// TIA Portal V17 export
// export: Created 2023-02-14T02:49:12.4327094Z, ExportSetting WithDefaults, DisplayName Totally Integrated Automation Portal, DisplayVersion V17, DisplayName TIA Portal Openness, DisplayVersion V17, DisplayName TIA Portal Teamcenter Gateway, DisplayVersion V17, DisplayName TIA Portal Version Control Interface, DisplayVersion V17, DisplayName SINAMICS Startdrive Advanced, DisplayVersion V17, DisplayName SINAMICS Startdrive G130, G150, S120, S150, SINAMICS MV, S210, DisplayVersion V17, DisplayName SINAMICS Startdrive G110M, G120, G120C, G120D, G120P, G115D, DisplayVersion V17, DisplayName STEP 7 Professional, DisplayVersion V17, DisplayName STEP 7 Safety, DisplayVersion V17, DisplayName WinCC Professional, DisplayVersion V17
FUNCTION "Comm" : Void   // FC7, LAD
{ S7_Optimized_Access := 'TRUE' }
VERSION : 0.1
// stored: AutoNumber true, IsIECCheckEnabled false, SetENOAutomatically false, UDAEnableTagReadback false
   VAR_TEMP   // added for the SCL form of the ladder/FBD networks
      _s5time1 : S5Time;
      _s5time2 : S5Time;
      _w1 : Bool;
   END_VAR
BEGIN

REGION Network 1: THE1 Heat Beat
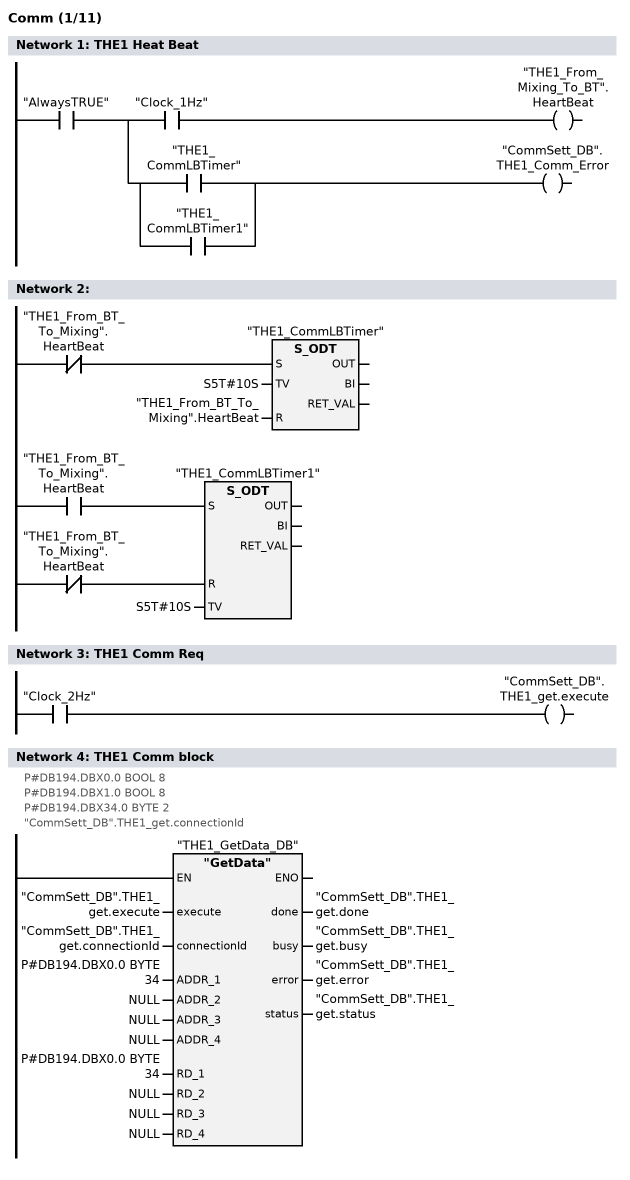
   RUNG wire#powerrail
      Contact( "AlwaysTRUE" )
      wire#w1
      Contact( "Clock_1Hz" )
      Coil( "THE1_From_Mixing_To_BT".HeartBeat )
   END_RUNG
   RUNG wire#w1
      Contact( "THE1_CommLBTimer" )
      wire#w2
      Coil( "CommSett_DB".THE1_Comm_Error )
   END_RUNG
   RUNG wire#w1
      Contact( "THE1_CommLBTimer1" )
   END_RUNG wire#w2
   // the same network as SCL:
   "THE1_From_Mixing_To_BT".HeartBeat := "AlwaysTRUE" AND "Clock_1Hz";
   "CommSett_DB".THE1_Comm_Error := "AlwaysTRUE" AND ("THE1_CommLBTimer" OR "THE1_CommLBTimer1");
END_REGION

REGION Network 2
   RUNG wire#powerrail
      I_Contact( "THE1_From_BT_To_Mixing".HeartBeat )
      S_ODT(T_NO := "THE1_CommLBTimer", TV := S5T#10S, R := "THE1_From_BT_To_Mixing".HeartBeat, BI =>, RET_VAL =>)
   END_RUNG
   RUNG wire#powerrail
      Contact( "THE1_From_BT_To_Mixing".HeartBeat )
      S_ODT(T_NO := "THE1_CommLBTimer1", R := wire#w1, TV := S5T#10S, BI =>, RET_VAL =>)
   END_RUNG
   RUNG wire#powerrail
      I_Contact( "THE1_From_BT_To_Mixing".HeartBeat )
   END_RUNG wire#w1
   // the same network as SCL:
   #_s5time1 := S_ODT(T_NO := "THE1_CommLBTimer",
                      S := NOT "THE1_From_BT_To_Mixing".HeartBeat,
                      TV := S5T#10S,
                      R := "THE1_From_BT_To_Mixing".HeartBeat);
   #_s5time2 := S_ODT(T_NO := "THE1_CommLBTimer1",
                      S := "THE1_From_BT_To_Mixing".HeartBeat,
                      R := NOT "THE1_From_BT_To_Mixing".HeartBeat,
                      TV := S5T#10S);
END_REGION

REGION Network 3: THE1 Comm Req
   RUNG wire#powerrail
      Contact( "Clock_2Hz" )
      Coil( "CommSett_DB".THE1_get.execute )
   END_RUNG
   // the same network as SCL:
   "CommSett_DB".THE1_get.execute := "Clock_2Hz";
END_REGION

REGION Network 4: THE1 Comm block
   // P#DB194.DBX0.0 BOOL 8
   // P#DB194.DBX1.0 BOOL 8
   // P#DB194.DBX34.0 BYTE 2
   // "CommSett_DB".THE1_get.connectionId
   RUNG wire#powerrail
      "THE1_GetData_DB"(execute := "CommSett_DB".THE1_get.execute, connectionId := "CommSett_DB".THE1_get.connectionId, ADDR_1 := P#DB194.DBX0.0 BYTE 34, ADDR_2 := NULL, ADDR_3 := NULL, ADDR_4 := NULL, RD_1 := P#DB194.DBX0.0 BYTE 34, RD_2 := NULL, RD_3 := NULL, RD_4 := NULL, done => "CommSett_DB".THE1_get.done, busy => "CommSett_DB".THE1_get.busy, error => "CommSett_DB".THE1_get.error, status => "CommSett_DB".THE1_get.status)
   END_RUNG
   // the same network as SCL:
   "THE1_GetData_DB"(execute := "CommSett_DB".THE1_get.execute,   // "GetData"
                     connectionId := "CommSett_DB".THE1_get.connectionId,
                     ADDR_1 := P#DB194.DBX0.0 BYTE 34,
                     ADDR_2 := NULL,
                     ADDR_3 := NULL,
                     ADDR_4 := NULL,
                     RD_1 := P#DB194.DBX0.0 BYTE 34,
                     RD_2 := NULL,
                     RD_3 := NULL,
                     RD_4 := NULL,
                     done => "CommSett_DB".THE1_get.done,
                     busy => "CommSett_DB".THE1_get.busy,
                     error => "CommSett_DB".THE1_get.error,
                     status => "CommSett_DB".THE1_get.status);
END_REGION

REGION Network 5
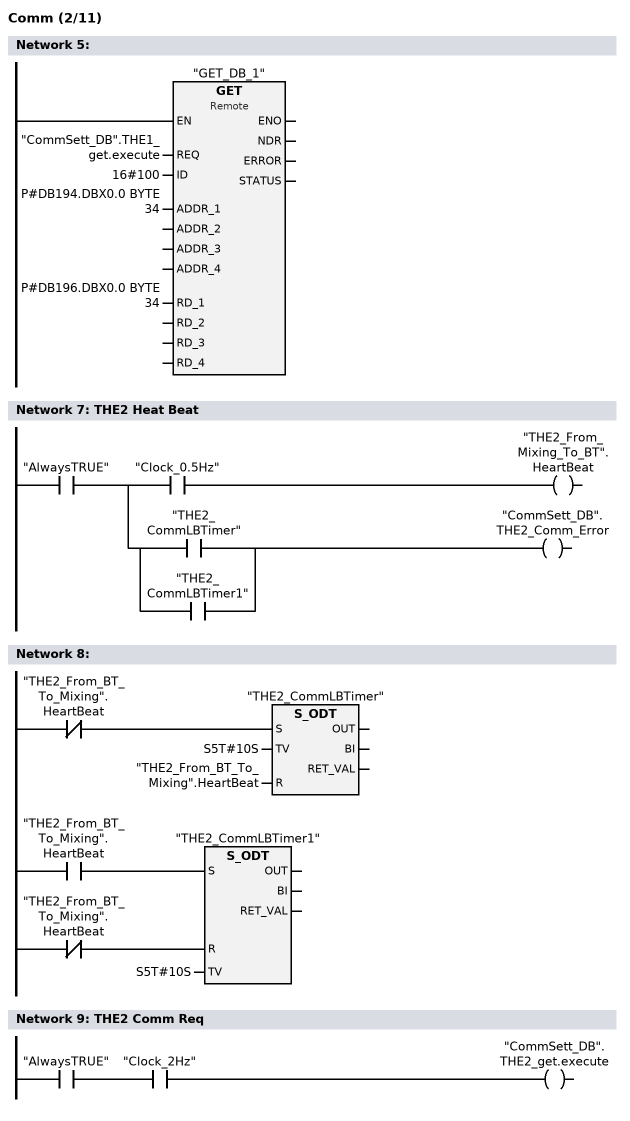
   RUNG wire#powerrail
      { S7_Templates := "[remote_type := Remote, local_type := Variant]" } "GET_DB_1".GET(REQ := "CommSett_DB".THE1_get.execute, ID := 16#100, ADDR_1 := P#DB194.DBX0.0 BYTE 34, ADDR_2 :=, ADDR_3 :=, ADDR_4 :=, RD_1 := P#DB196.DBX0.0 BYTE 34, RD_2 :=, RD_3 :=, RD_4 :=, NDR =>, ERROR =>, STATUS =>)
   END_RUNG
   // the same network as SCL:
   "GET_DB_1"(REQ := "CommSett_DB".THE1_get.execute,   // GET
              ID := 16#100,
              ADDR_1 := P#DB194.DBX0.0 BYTE 34,
              RD_1 := P#DB196.DBX0.0 BYTE 34);
END_REGION

REGION Network 6 (SCL): THE1 Comm Diag
   IF ("CommSett_DB".THE1_get.done = TRUE
       OR "CommSett_DB".THE1_get.error = true)
       AND "CommSett_DB".THE1_get.execute = TRUE
   THEN
       "CommSett_DB".THE1_get.execute := false;
       "CommSett_DB".THE1_diagnostic.statusGet := "CommSett_DB".THE1_get.status;
   END_IF;
END_REGION

REGION Network 7: THE2 Heat Beat
   RUNG wire#powerrail
      Contact( "AlwaysTRUE" )
      wire#w1
      Contact( "Clock_0.5Hz" )
      Coil( "THE2_From_Mixing_To_BT".HeartBeat )
   END_RUNG
   RUNG wire#w1
      Contact( "THE2_CommLBTimer" )
      wire#w2
      Coil( "CommSett_DB".THE2_Comm_Error )
   END_RUNG
   RUNG wire#w1
      Contact( "THE2_CommLBTimer1" )
   END_RUNG wire#w2
   // the same network as SCL:
   "THE2_From_Mixing_To_BT".HeartBeat := "AlwaysTRUE" AND "Clock_0.5Hz";
   "CommSett_DB".THE2_Comm_Error := "AlwaysTRUE" AND ("THE2_CommLBTimer" OR "THE2_CommLBTimer1");
END_REGION

REGION Network 8
   RUNG wire#powerrail
      I_Contact( "THE2_From_BT_To_Mixing".HeartBeat )
      S_ODT(T_NO := "THE2_CommLBTimer", TV := S5T#10S, R := "THE2_From_BT_To_Mixing".HeartBeat, BI =>, RET_VAL =>)
   END_RUNG
   RUNG wire#powerrail
      Contact( "THE2_From_BT_To_Mixing".HeartBeat )
      S_ODT(T_NO := "THE2_CommLBTimer1", R := wire#w1, TV := S5T#10S, BI =>, RET_VAL =>)
   END_RUNG
   RUNG wire#powerrail
      I_Contact( "THE2_From_BT_To_Mixing".HeartBeat )
   END_RUNG wire#w1
   // the same network as SCL:
   #_s5time1 := S_ODT(T_NO := "THE2_CommLBTimer",
                      S := NOT "THE2_From_BT_To_Mixing".HeartBeat,
                      TV := S5T#10S,
                      R := "THE2_From_BT_To_Mixing".HeartBeat);
   #_s5time2 := S_ODT(T_NO := "THE2_CommLBTimer1",
                      S := "THE2_From_BT_To_Mixing".HeartBeat,
                      R := NOT "THE2_From_BT_To_Mixing".HeartBeat,
                      TV := S5T#10S);
END_REGION

REGION Network 9: THE2 Comm Req
   RUNG wire#powerrail
      Contact( "AlwaysTRUE" )
      Contact( "Clock_2Hz" )
      Coil( "CommSett_DB".THE2_get.execute )
   END_RUNG
   // the same network as SCL:
   "CommSett_DB".THE2_get.execute := "AlwaysTRUE" AND "Clock_2Hz";
END_REGION

REGION Network 10: THE2 Comm block
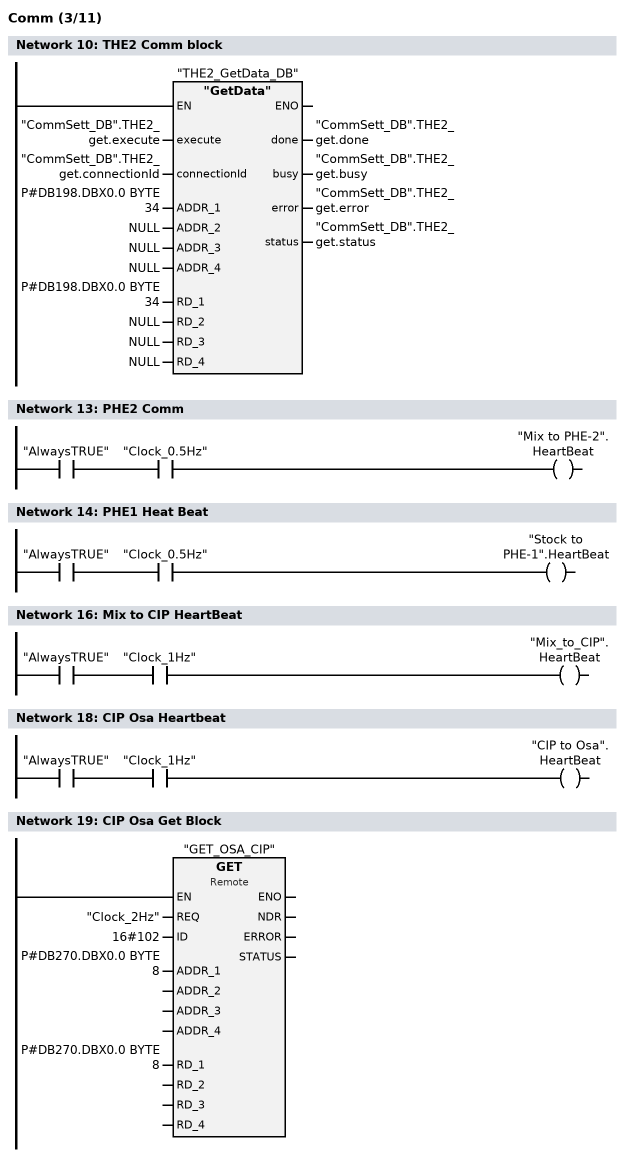
   RUNG wire#powerrail
      "THE2_GetData_DB"(execute := "CommSett_DB".THE2_get.execute, connectionId := "CommSett_DB".THE2_get.connectionId, ADDR_1 := P#DB198.DBX0.0 BYTE 34, ADDR_2 := NULL, ADDR_3 := NULL, ADDR_4 := NULL, RD_1 := P#DB198.DBX0.0 BYTE 34, RD_2 := NULL, RD_3 := NULL, RD_4 := NULL, done => "CommSett_DB".THE2_get.done, busy => "CommSett_DB".THE2_get.busy, error => "CommSett_DB".THE2_get.error, status => "CommSett_DB".THE2_get.status)
   END_RUNG
   // the same network as SCL:
   "THE2_GetData_DB"(execute := "CommSett_DB".THE2_get.execute,   // "GetData"
                     connectionId := "CommSett_DB".THE2_get.connectionId,
                     ADDR_1 := P#DB198.DBX0.0 BYTE 34,
                     ADDR_2 := NULL,
                     ADDR_3 := NULL,
                     ADDR_4 := NULL,
                     RD_1 := P#DB198.DBX0.0 BYTE 34,
                     RD_2 := NULL,
                     RD_3 := NULL,
                     RD_4 := NULL,
                     done => "CommSett_DB".THE2_get.done,
                     busy => "CommSett_DB".THE2_get.busy,
                     error => "CommSett_DB".THE2_get.error,
                     status => "CommSett_DB".THE2_get.status);
END_REGION

REGION Network 11 (SCL): THE2 Comm Diag
   IF ("CommSett_DB".THE2_get.done = TRUE
       OR "CommSett_DB".THE2_get.error = true)
       AND "CommSett_DB".THE2_get.execute = TRUE
   THEN
       "CommSett_DB".THE2_get.execute := false;
       "CommSett_DB".THE2_diagnostic.statusGet := "CommSett_DB".THE2_get.status;
   END_IF;
END_REGION

REGION Network 13: PHE2 Comm
   RUNG wire#powerrail
      Contact( "AlwaysTRUE" )
      Contact( "Clock_0.5Hz" )
      Coil( "Mix to PHE-2".HeartBeat )
   END_RUNG
   // the same network as SCL:
   "Mix to PHE-2".HeartBeat := "AlwaysTRUE" AND "Clock_0.5Hz";
END_REGION

REGION Network 14: PHE1 Heat Beat
   RUNG wire#powerrail
      Contact( "AlwaysTRUE" )
      Contact( "Clock_0.5Hz" )
      Coil( "Stock to PHE-1".HeartBeat )
   END_RUNG
   // the same network as SCL:
   "Stock to PHE-1".HeartBeat := "AlwaysTRUE" AND "Clock_0.5Hz";
END_REGION

REGION Network 16: Mix to CIP HeartBeat
   RUNG wire#powerrail
      Contact( "AlwaysTRUE" )
      Contact( "Clock_1Hz" )
      Coil( "Mix_to_CIP".HeartBeat )
   END_RUNG
   // the same network as SCL:
   "Mix_to_CIP".HeartBeat := "AlwaysTRUE" AND "Clock_1Hz";
END_REGION

REGION Network 18: CIP Osa Heartbeat
   RUNG wire#powerrail
      Contact( "AlwaysTRUE" )
      Contact( "Clock_1Hz" )
      Coil( "CIP to Osa".HeartBeat )
   END_RUNG
   // the same network as SCL:
   "CIP to Osa".HeartBeat := "AlwaysTRUE" AND "Clock_1Hz";
END_REGION

REGION Network 19: CIP Osa Get Block
   RUNG wire#powerrail
      { S7_Templates := "[remote_type := Remote, local_type := Variant]" } "GET_OSA_CIP".GET(REQ := "Clock_2Hz", ID := 16#102, ADDR_1 := P#DB270.DBX0.0 BYTE 8, ADDR_2 :=, ADDR_3 :=, ADDR_4 :=, RD_1 := P#DB270.DBX0.0 BYTE 8, RD_2 :=, RD_3 :=, RD_4 :=, NDR =>, ERROR =>, STATUS =>)
   END_RUNG
   // the same network as SCL:
   "GET_OSA_CIP"(REQ := "Clock_2Hz",   // GET
                 ID := 16#102,
                 ADDR_1 := P#DB270.DBX0.0 BYTE 8,
                 RD_1 := P#DB270.DBX0.0 BYTE 8);
END_REGION

REGION Network 20: CIP Osa Put Block
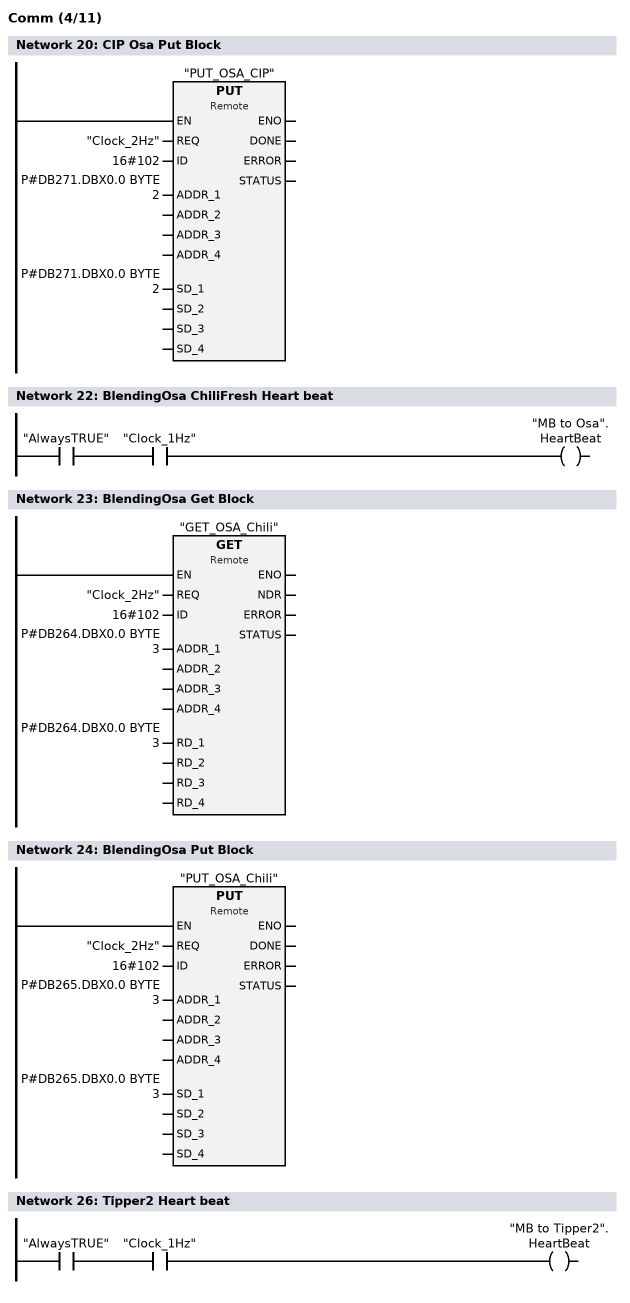
   RUNG wire#powerrail
      { S7_Templates := "[remote_type := Remote, local_type := Variant]" } "PUT_OSA_CIP".PUT(REQ := "Clock_2Hz", ID := 16#102, ADDR_1 := P#DB271.DBX0.0 BYTE 2, ADDR_2 :=, ADDR_3 :=, ADDR_4 :=, SD_1 := P#DB271.DBX0.0 BYTE 2, SD_2 :=, SD_3 :=, SD_4 :=, DONE =>, ERROR =>, STATUS =>)
   END_RUNG
   // the same network as SCL:
   "PUT_OSA_CIP"(REQ := "Clock_2Hz",   // PUT
                 ID := 16#102,
                 ADDR_1 := P#DB271.DBX0.0 BYTE 2,
                 SD_1 := P#DB271.DBX0.0 BYTE 2);
END_REGION

REGION Network 22: BlendingOsa ChiliFresh Heart beat
   RUNG wire#powerrail
      Contact( "AlwaysTRUE" )
      Contact( "Clock_1Hz" )
      Coil( "MB to Osa".HeartBeat )
   END_RUNG
   // the same network as SCL:
   "MB to Osa".HeartBeat := "AlwaysTRUE" AND "Clock_1Hz";
END_REGION

REGION Network 23: BlendingOsa Get Block
   RUNG wire#powerrail
      { S7_Templates := "[remote_type := Remote, local_type := Variant]" } "GET_OSA_Chili".GET(REQ := "Clock_2Hz", ID := 16#102, ADDR_1 := P#DB264.DBX0.0 BYTE 3, ADDR_2 :=, ADDR_3 :=, ADDR_4 :=, RD_1 := P#DB264.DBX0.0 BYTE 3, RD_2 :=, RD_3 :=, RD_4 :=, NDR =>, ERROR =>, STATUS =>)
   END_RUNG
   // the same network as SCL:
   "GET_OSA_Chili"(REQ := "Clock_2Hz",   // GET
                   ID := 16#102,
                   ADDR_1 := P#DB264.DBX0.0 BYTE 3,
                   RD_1 := P#DB264.DBX0.0 BYTE 3);
END_REGION

REGION Network 24: BlendingOsa Put Block
   RUNG wire#powerrail
      { S7_Templates := "[remote_type := Remote, local_type := Variant]" } "PUT_OSA_Chili".PUT(REQ := "Clock_2Hz", ID := 16#102, ADDR_1 := P#DB265.DBX0.0 BYTE 3, ADDR_2 :=, ADDR_3 :=, ADDR_4 :=, SD_1 := P#DB265.DBX0.0 BYTE 3, SD_2 :=, SD_3 :=, SD_4 :=, DONE =>, ERROR =>, STATUS =>)
   END_RUNG
   // the same network as SCL:
   "PUT_OSA_Chili"(REQ := "Clock_2Hz",   // PUT
                   ID := 16#102,
                   ADDR_1 := P#DB265.DBX0.0 BYTE 3,
                   SD_1 := P#DB265.DBX0.0 BYTE 3);
END_REGION

REGION Network 26: Tipper2 Heart beat
   RUNG wire#powerrail
      Contact( "AlwaysTRUE" )
      Contact( "Clock_1Hz" )
      Coil( "MB to Tipper2".HeartBeat )
   END_RUNG
   // the same network as SCL:
   "MB to Tipper2".HeartBeat := "AlwaysTRUE" AND "Clock_1Hz";
END_REGION

REGION Network 27: Tipper2 Get Block
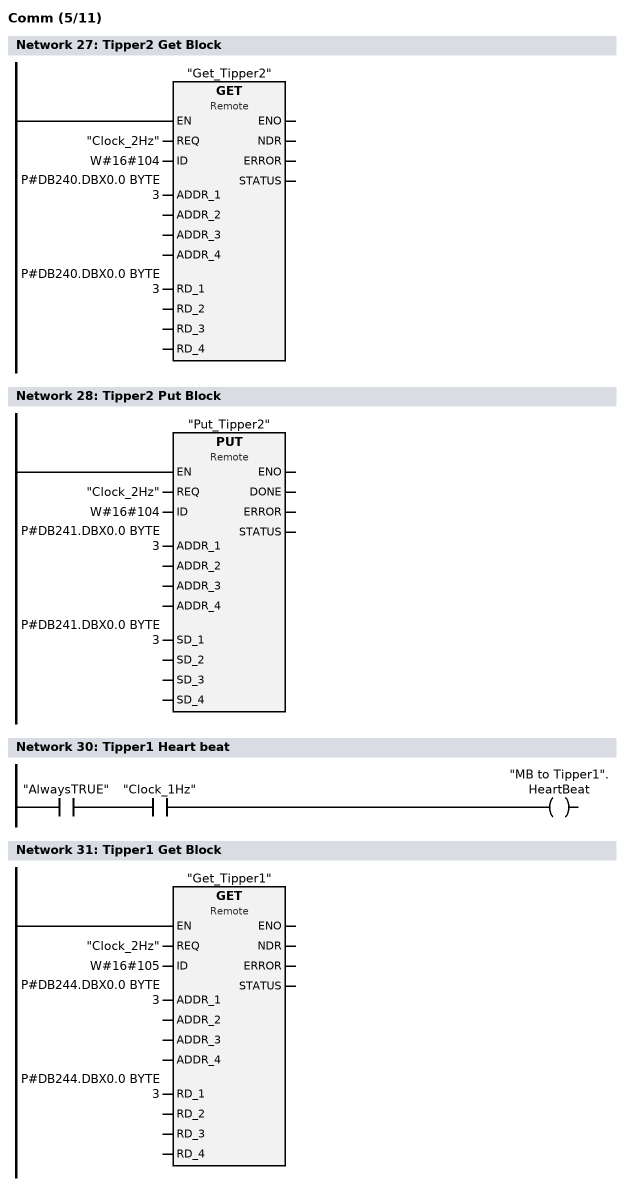
   RUNG wire#powerrail
      { S7_Templates := "[remote_type := Remote, local_type := Variant]" } "Get_Tipper2".GET(REQ := "Clock_2Hz", ID := W#16#104, ADDR_1 := P#DB240.DBX0.0 BYTE 3, ADDR_2 :=, ADDR_3 :=, ADDR_4 :=, RD_1 := P#DB240.DBX0.0 BYTE 3, RD_2 :=, RD_3 :=, RD_4 :=, NDR =>, ERROR =>, STATUS =>)
   END_RUNG
   // the same network as SCL:
   "Get_Tipper2"(REQ := "Clock_2Hz",   // GET
                 ID := W#16#104,
                 ADDR_1 := P#DB240.DBX0.0 BYTE 3,
                 RD_1 := P#DB240.DBX0.0 BYTE 3);
END_REGION

REGION Network 28: Tipper2 Put Block
   RUNG wire#powerrail
      { S7_Templates := "[remote_type := Remote, local_type := Variant]" } "Put_Tipper2".PUT(REQ := "Clock_2Hz", ID := W#16#104, ADDR_1 := P#DB241.DBX0.0 BYTE 3, ADDR_2 :=, ADDR_3 :=, ADDR_4 :=, SD_1 := P#DB241.DBX0.0 BYTE 3, SD_2 :=, SD_3 :=, SD_4 :=, DONE =>, ERROR =>, STATUS =>)
   END_RUNG
   // the same network as SCL:
   "Put_Tipper2"(REQ := "Clock_2Hz",   // PUT
                 ID := W#16#104,
                 ADDR_1 := P#DB241.DBX0.0 BYTE 3,
                 SD_1 := P#DB241.DBX0.0 BYTE 3);
END_REGION

REGION Network 30: Tipper1 Heart beat
   RUNG wire#powerrail
      Contact( "AlwaysTRUE" )
      Contact( "Clock_1Hz" )
      Coil( "MB to Tipper1".HeartBeat )
   END_RUNG
   // the same network as SCL:
   "MB to Tipper1".HeartBeat := "AlwaysTRUE" AND "Clock_1Hz";
END_REGION

REGION Network 31: Tipper1 Get Block
   RUNG wire#powerrail
      { S7_Templates := "[remote_type := Remote, local_type := Variant]" } "Get_Tipper1".GET(REQ := "Clock_2Hz", ID := W#16#105, ADDR_1 := P#DB244.DBX0.0 BYTE 3, ADDR_2 :=, ADDR_3 :=, ADDR_4 :=, RD_1 := P#DB244.DBX0.0 BYTE 3, RD_2 :=, RD_3 :=, RD_4 :=, NDR =>, ERROR =>, STATUS =>)
   END_RUNG
   // the same network as SCL:
   "Get_Tipper1"(REQ := "Clock_2Hz",   // GET
                 ID := W#16#105,
                 ADDR_1 := P#DB244.DBX0.0 BYTE 3,
                 RD_1 := P#DB244.DBX0.0 BYTE 3);
END_REGION

REGION Network 32: Tipper1 Put Block
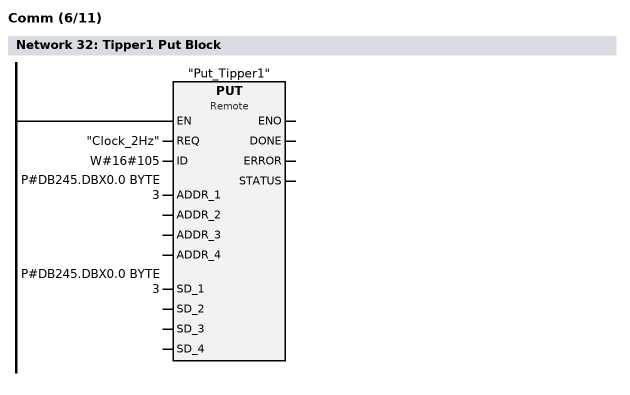
   RUNG wire#powerrail
      { S7_Templates := "[remote_type := Remote, local_type := Variant]" } "Put_Tipper1".PUT(REQ := "Clock_2Hz", ID := W#16#105, ADDR_1 := P#DB245.DBX0.0 BYTE 3, ADDR_2 :=, ADDR_3 :=, ADDR_4 :=, SD_1 := P#DB245.DBX0.0 BYTE 3, SD_2 :=, SD_3 :=, SD_4 :=, DONE =>, ERROR =>, STATUS =>)
   END_RUNG
   // the same network as SCL:
   "Put_Tipper1"(REQ := "Clock_2Hz",   // PUT
                 ID := W#16#105,
                 ADDR_1 := P#DB245.DBX0.0 BYTE 3,
                 SD_1 := P#DB245.DBX0.0 BYTE 3);
END_REGION

REGION Network 34: CIP Enable for Tipper 1, Tipper 2, and Blend OSA
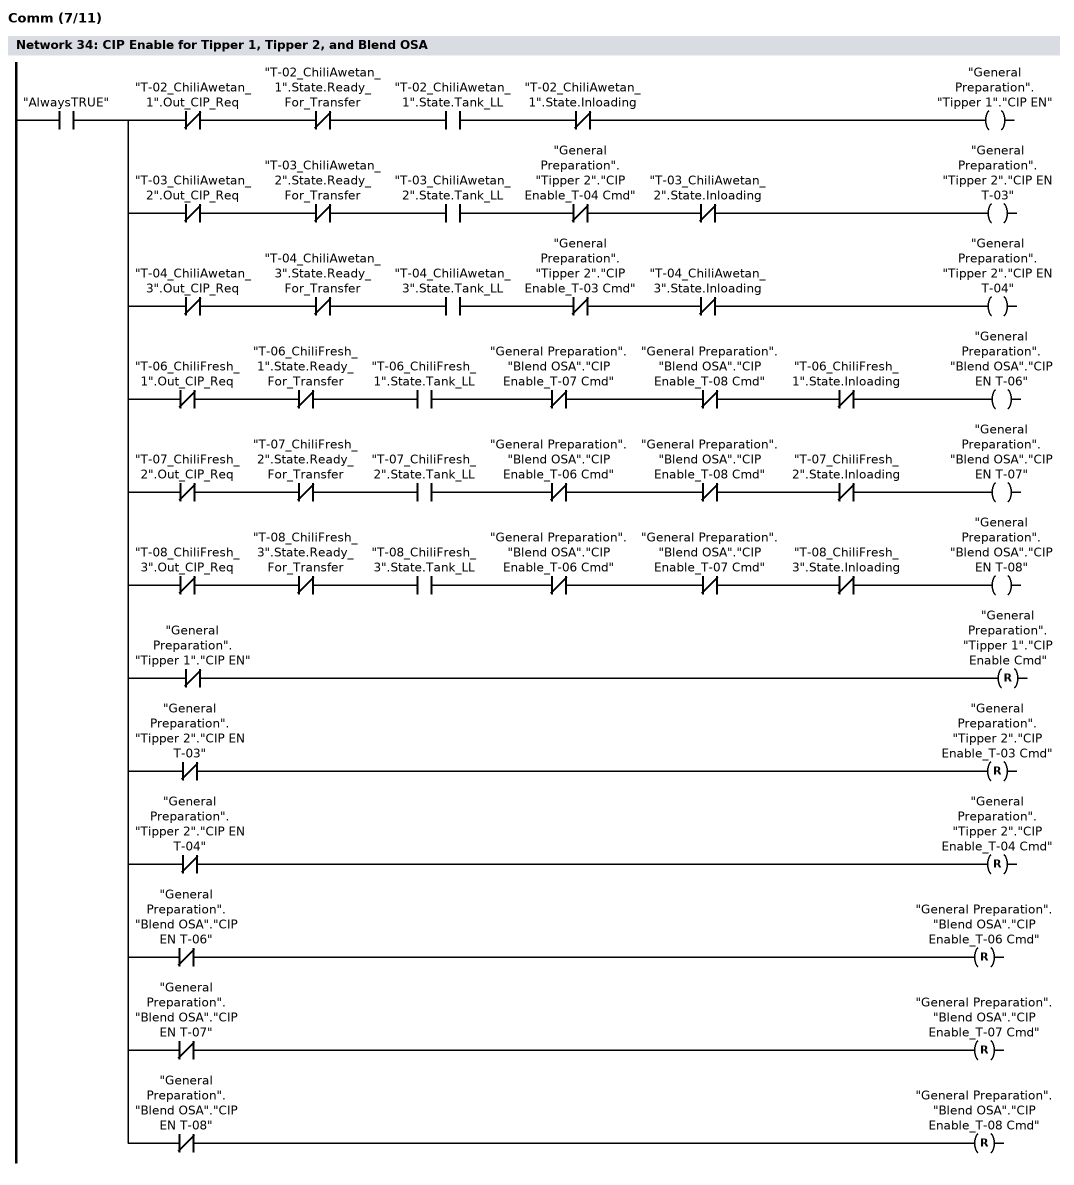
   RUNG wire#powerrail
      Contact( "AlwaysTRUE" )
      wire#w1
      I_Contact( "T-02_ChiliAwetan_1".Out_CIP_Req )
      I_Contact( "T-02_ChiliAwetan_1".State.Ready_For_Transfer )
      Contact( "T-02_ChiliAwetan_1".State.Tank_LL )
      I_Contact( "T-02_ChiliAwetan_1".State.Inloading )
      Coil( "General Preparation"."Tipper 1"."CIP EN" )
   END_RUNG
   RUNG wire#w1
      I_Contact( "T-03_ChiliAwetan_2".Out_CIP_Req )
      I_Contact( "T-03_ChiliAwetan_2".State.Ready_For_Transfer )
      Contact( "T-03_ChiliAwetan_2".State.Tank_LL )
      I_Contact( "General Preparation"."Tipper 2"."CIP Enable_T-04 Cmd" )
      I_Contact( "T-03_ChiliAwetan_2".State.Inloading )
      Coil( "General Preparation"."Tipper 2"."CIP EN T-03" )
   END_RUNG
   RUNG wire#w1
      I_Contact( "T-04_ChiliAwetan_3".Out_CIP_Req )
      I_Contact( "T-04_ChiliAwetan_3".State.Ready_For_Transfer )
      Contact( "T-04_ChiliAwetan_3".State.Tank_LL )
      I_Contact( "General Preparation"."Tipper 2"."CIP Enable_T-03 Cmd" )
      I_Contact( "T-04_ChiliAwetan_3".State.Inloading )
      Coil( "General Preparation"."Tipper 2"."CIP EN T-04" )
   END_RUNG
   RUNG wire#w1
      I_Contact( "T-06_ChiliFresh_1".Out_CIP_Req )
      I_Contact( "T-06_ChiliFresh_1".State.Ready_For_Transfer )
      Contact( "T-06_ChiliFresh_1".State.Tank_LL )
      I_Contact( "General Preparation"."Blend OSA"."CIP Enable_T-07 Cmd" )
      I_Contact( "General Preparation"."Blend OSA"."CIP Enable_T-08 Cmd" )
      I_Contact( "T-06_ChiliFresh_1".State.Inloading )
      Coil( "General Preparation"."Blend OSA"."CIP EN T-06" )
   END_RUNG
   RUNG wire#w1
      I_Contact( "T-07_ChiliFresh_2".Out_CIP_Req )
      I_Contact( "T-07_ChiliFresh_2".State.Ready_For_Transfer )
      Contact( "T-07_ChiliFresh_2".State.Tank_LL )
      I_Contact( "General Preparation"."Blend OSA"."CIP Enable_T-06 Cmd" )
      I_Contact( "General Preparation"."Blend OSA"."CIP Enable_T-08 Cmd" )
      I_Contact( "T-07_ChiliFresh_2".State.Inloading )
      Coil( "General Preparation"."Blend OSA"."CIP EN T-07" )
   END_RUNG
   RUNG wire#w1
      I_Contact( "T-08_ChiliFresh_3".Out_CIP_Req )
      I_Contact( "T-08_ChiliFresh_3".State.Ready_For_Transfer )
      Contact( "T-08_ChiliFresh_3".State.Tank_LL )
      I_Contact( "General Preparation"."Blend OSA"."CIP Enable_T-06 Cmd" )
      I_Contact( "General Preparation"."Blend OSA"."CIP Enable_T-07 Cmd" )
      I_Contact( "T-08_ChiliFresh_3".State.Inloading )
      Coil( "General Preparation"."Blend OSA"."CIP EN T-08" )
   END_RUNG
   RUNG wire#w1
      I_Contact( "General Preparation"."Tipper 1"."CIP EN" )
      R_Coil( "General Preparation"."Tipper 1"."CIP Enable Cmd" )
   END_RUNG
   RUNG wire#w1
      I_Contact( "General Preparation"."Tipper 2"."CIP EN T-03" )
      R_Coil( "General Preparation"."Tipper 2"."CIP Enable_T-03 Cmd" )
   END_RUNG
   RUNG wire#w1
      I_Contact( "General Preparation"."Tipper 2"."CIP EN T-04" )
      R_Coil( "General Preparation"."Tipper 2"."CIP Enable_T-04 Cmd" )
   END_RUNG
   RUNG wire#w1
      I_Contact( "General Preparation"."Blend OSA"."CIP EN T-06" )
      R_Coil( "General Preparation"."Blend OSA"."CIP Enable_T-06 Cmd" )
   END_RUNG
   RUNG wire#w1
      I_Contact( "General Preparation"."Blend OSA"."CIP EN T-07" )
      R_Coil( "General Preparation"."Blend OSA"."CIP Enable_T-07 Cmd" )
   END_RUNG
   RUNG wire#w1
      I_Contact( "General Preparation"."Blend OSA"."CIP EN T-08" )
      R_Coil( "General Preparation"."Blend OSA"."CIP Enable_T-08 Cmd" )
   END_RUNG
   // the same network as SCL:
   "General Preparation"."Tipper 1"."CIP EN" := "AlwaysTRUE" AND NOT "T-02_ChiliAwetan_1".Out_CIP_Req AND NOT "T-02_ChiliAwetan_1".State.Ready_For_Transfer AND "T-02_ChiliAwetan_1".State.Tank_LL AND NOT "T-02_ChiliAwetan_1".State.Inloading;
   "General Preparation"."Tipper 2"."CIP EN T-03" := "AlwaysTRUE" AND NOT "T-03_ChiliAwetan_2".Out_CIP_Req AND NOT "T-03_ChiliAwetan_2".State.Ready_For_Transfer AND "T-03_ChiliAwetan_2".State.Tank_LL AND NOT "General Preparation"."Tipper 2"."CIP Enable_T-04 Cmd" AND NOT "T-03_ChiliAwetan_2".State.Inloading;
   "General Preparation"."Tipper 2"."CIP EN T-04" := "AlwaysTRUE" AND NOT "T-04_ChiliAwetan_3".Out_CIP_Req AND NOT "T-04_ChiliAwetan_3".State.Ready_For_Transfer AND "T-04_ChiliAwetan_3".State.Tank_LL AND NOT "General Preparation"."Tipper 2"."CIP Enable_T-03 Cmd" AND NOT "T-04_ChiliAwetan_3".State.Inloading;
   "General Preparation"."Blend OSA"."CIP EN T-06" := "AlwaysTRUE" AND NOT "T-06_ChiliFresh_1".Out_CIP_Req AND NOT "T-06_ChiliFresh_1".State.Ready_For_Transfer AND "T-06_ChiliFresh_1".State.Tank_LL AND NOT "General Preparation"."Blend OSA"."CIP Enable_T-07 Cmd" AND NOT "General Preparation"."Blend OSA"."CIP Enable_T-08 Cmd" AND NOT "T-06_ChiliFresh_1".State.Inloading;
   "General Preparation"."Blend OSA"."CIP EN T-07" := "AlwaysTRUE" AND NOT "T-07_ChiliFresh_2".Out_CIP_Req AND NOT "T-07_ChiliFresh_2".State.Ready_For_Transfer AND "T-07_ChiliFresh_2".State.Tank_LL AND NOT "General Preparation"."Blend OSA"."CIP Enable_T-06 Cmd" AND NOT "General Preparation"."Blend OSA"."CIP Enable_T-08 Cmd" AND NOT "T-07_ChiliFresh_2".State.Inloading;
   "General Preparation"."Blend OSA"."CIP EN T-08" := "AlwaysTRUE" AND NOT "T-08_ChiliFresh_3".Out_CIP_Req AND NOT "T-08_ChiliFresh_3".State.Ready_For_Transfer AND "T-08_ChiliFresh_3".State.Tank_LL AND NOT "General Preparation"."Blend OSA"."CIP Enable_T-06 Cmd" AND NOT "General Preparation"."Blend OSA"."CIP Enable_T-07 Cmd" AND NOT "T-08_ChiliFresh_3".State.Inloading;
   IF "AlwaysTRUE" AND NOT "General Preparation"."Tipper 1"."CIP EN" THEN
       "General Preparation"."Tipper 1"."CIP Enable Cmd" := FALSE;
   END_IF;
   IF "AlwaysTRUE" AND NOT "General Preparation"."Tipper 2"."CIP EN T-03" THEN
       "General Preparation"."Tipper 2"."CIP Enable_T-03 Cmd" := FALSE;
   END_IF;
   IF "AlwaysTRUE" AND NOT "General Preparation"."Tipper 2"."CIP EN T-04" THEN
       "General Preparation"."Tipper 2"."CIP Enable_T-04 Cmd" := FALSE;
   END_IF;
   IF "AlwaysTRUE" AND NOT "General Preparation"."Blend OSA"."CIP EN T-06" THEN
       "General Preparation"."Blend OSA"."CIP Enable_T-06 Cmd" := FALSE;
   END_IF;
   IF "AlwaysTRUE" AND NOT "General Preparation"."Blend OSA"."CIP EN T-07" THEN
       "General Preparation"."Blend OSA"."CIP Enable_T-07 Cmd" := FALSE;
   END_IF;
   IF "AlwaysTRUE" AND NOT "General Preparation"."Blend OSA"."CIP EN T-08" THEN
       "General Preparation"."Blend OSA"."CIP Enable_T-08 Cmd" := FALSE;
   END_IF;
END_REGION

REGION Network 35: CIP Request Status for Tipper 1, TIpper 2, Blend OSA
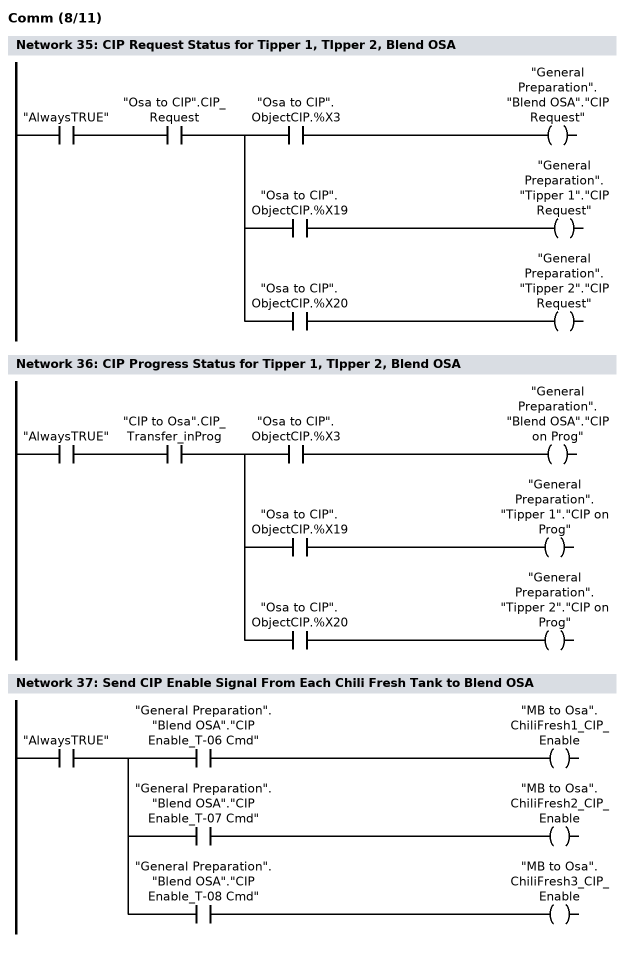
   RUNG wire#powerrail
      Contact( "AlwaysTRUE" )
      Contact( "Osa to CIP".CIP_Request )
      wire#w1
      Contact( "Osa to CIP".ObjectCIP.%X3 )
      Coil( "General Preparation"."Blend OSA"."CIP Request" )
   END_RUNG
   RUNG wire#w1
      Contact( "Osa to CIP".ObjectCIP.%X19 )
      Coil( "General Preparation"."Tipper 1"."CIP Request" )
   END_RUNG
   RUNG wire#w1
      Contact( "Osa to CIP".ObjectCIP.%X20 )
      Coil( "General Preparation"."Tipper 2"."CIP Request" )
   END_RUNG
   // the same network as SCL:
   #_w1 := "AlwaysTRUE" AND "Osa to CIP".CIP_Request;
   "General Preparation"."Blend OSA"."CIP Request" := #_w1 AND "Osa to CIP".ObjectCIP.%X3;
   "General Preparation"."Tipper 1"."CIP Request" := #_w1 AND "Osa to CIP".ObjectCIP.%X19;
   "General Preparation"."Tipper 2"."CIP Request" := #_w1 AND "Osa to CIP".ObjectCIP.%X20;
END_REGION

REGION Network 36: CIP Progress Status for Tipper 1, TIpper 2, Blend OSA
   RUNG wire#powerrail
      Contact( "AlwaysTRUE" )
      Contact( "CIP to Osa".CIP_Transfer_inProg )
      wire#w1
      Contact( "Osa to CIP".ObjectCIP.%X3 )
      Coil( "General Preparation"."Blend OSA"."CIP on Prog" )
   END_RUNG
   RUNG wire#w1
      Contact( "Osa to CIP".ObjectCIP.%X19 )
      Coil( "General Preparation"."Tipper 1"."CIP on Prog" )
   END_RUNG
   RUNG wire#w1
      Contact( "Osa to CIP".ObjectCIP.%X20 )
      Coil( "General Preparation"."Tipper 2"."CIP on Prog" )
   END_RUNG
   // the same network as SCL:
   #_w1 := "AlwaysTRUE" AND "CIP to Osa".CIP_Transfer_inProg;
   "General Preparation"."Blend OSA"."CIP on Prog" := #_w1 AND "Osa to CIP".ObjectCIP.%X3;
   "General Preparation"."Tipper 1"."CIP on Prog" := #_w1 AND "Osa to CIP".ObjectCIP.%X19;
   "General Preparation"."Tipper 2"."CIP on Prog" := #_w1 AND "Osa to CIP".ObjectCIP.%X20;
END_REGION

REGION Network 37: Send CIP Enable Signal From Each Chili Fresh Tank to Blend OSA
   RUNG wire#powerrail
      Contact( "AlwaysTRUE" )
      wire#w1
      Contact( "General Preparation"."Blend OSA"."CIP Enable_T-06 Cmd" )
      Coil( "MB to Osa".ChiliFresh1_CIP_Enable )
   END_RUNG
   RUNG wire#w1
      Contact( "General Preparation"."Blend OSA"."CIP Enable_T-07 Cmd" )
      Coil( "MB to Osa".ChiliFresh2_CIP_Enable )
   END_RUNG
   RUNG wire#w1
      Contact( "General Preparation"."Blend OSA"."CIP Enable_T-08 Cmd" )
      Coil( "MB to Osa".ChiliFresh3_CIP_Enable )
   END_RUNG
   // the same network as SCL:
   "MB to Osa".ChiliFresh1_CIP_Enable := "AlwaysTRUE" AND "General Preparation"."Blend OSA"."CIP Enable_T-06 Cmd";
   "MB to Osa".ChiliFresh2_CIP_Enable := "AlwaysTRUE" AND "General Preparation"."Blend OSA"."CIP Enable_T-07 Cmd";
   "MB to Osa".ChiliFresh3_CIP_Enable := "AlwaysTRUE" AND "General Preparation"."Blend OSA"."CIP Enable_T-08 Cmd";
END_REGION

REGION Network 38: Send Status CIP Preparation Running to OSA
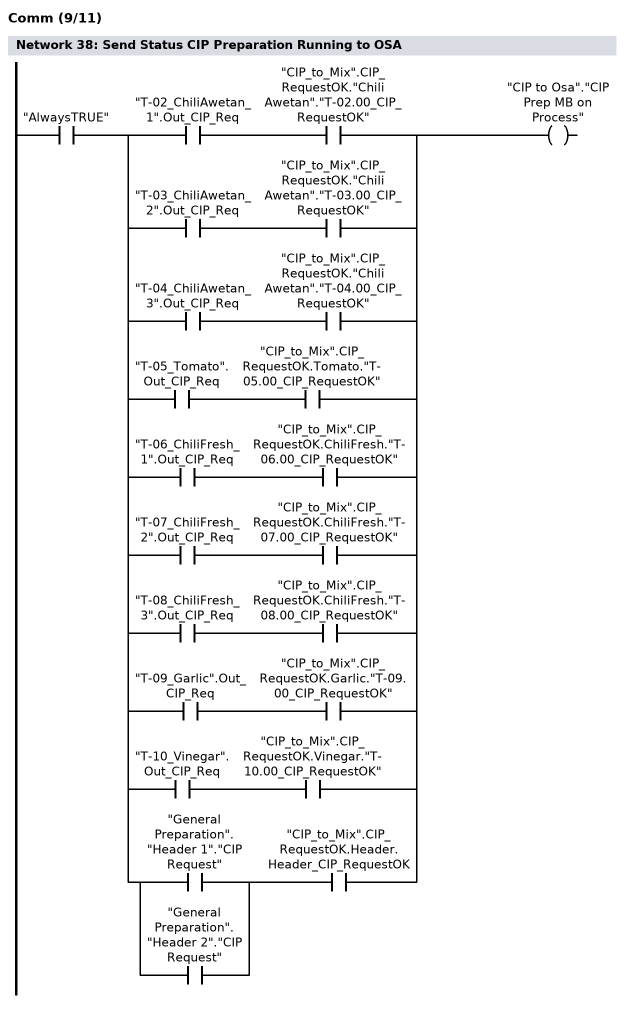
   RUNG wire#powerrail
      Contact( "AlwaysTRUE" )
      wire#w1
      Contact( "T-02_ChiliAwetan_1".Out_CIP_Req )
      Contact( "CIP_to_Mix".CIP_RequestOK."Chili Awetan"."T-02.00_CIP_RequestOK" )
      wire#w2
      Coil( "CIP to Osa"."CIP Prep MB on Process" )
   END_RUNG
   RUNG wire#w1
      Contact( "T-03_ChiliAwetan_2".Out_CIP_Req )
      Contact( "CIP_to_Mix".CIP_RequestOK."Chili Awetan"."T-03.00_CIP_RequestOK" )
   END_RUNG wire#w2
   RUNG wire#w1
      Contact( "T-04_ChiliAwetan_3".Out_CIP_Req )
      Contact( "CIP_to_Mix".CIP_RequestOK."Chili Awetan"."T-04.00_CIP_RequestOK" )
   END_RUNG wire#w2
   RUNG wire#w1
      Contact( "T-05_Tomato".Out_CIP_Req )
      Contact( "CIP_to_Mix".CIP_RequestOK.Tomato."T-05.00_CIP_RequestOK" )
   END_RUNG wire#w2
   RUNG wire#w1
      Contact( "T-06_ChiliFresh_1".Out_CIP_Req )
      Contact( "CIP_to_Mix".CIP_RequestOK.ChiliFresh."T-06.00_CIP_RequestOK" )
   END_RUNG wire#w2
   RUNG wire#w1
      Contact( "T-07_ChiliFresh_2".Out_CIP_Req )
      Contact( "CIP_to_Mix".CIP_RequestOK.ChiliFresh."T-07.00_CIP_RequestOK" )
   END_RUNG wire#w2
   RUNG wire#w1
      Contact( "T-08_ChiliFresh_3".Out_CIP_Req )
      Contact( "CIP_to_Mix".CIP_RequestOK.ChiliFresh."T-08.00_CIP_RequestOK" )
   END_RUNG wire#w2
   RUNG wire#w1
      Contact( "T-09_Garlic".Out_CIP_Req )
      Contact( "CIP_to_Mix".CIP_RequestOK.Garlic."T-09.00_CIP_RequestOK" )
   END_RUNG wire#w2
   RUNG wire#w1
      Contact( "T-10_Vinegar".Out_CIP_Req )
      Contact( "CIP_to_Mix".CIP_RequestOK.Vinegar."T-10.00_CIP_RequestOK" )
   END_RUNG wire#w2
   RUNG wire#w1
      Contact( "General Preparation"."Header 1"."CIP Request" )
      wire#w3
      Contact( "CIP_to_Mix".CIP_RequestOK.Header.Header_CIP_RequestOK )
   END_RUNG wire#w2
   RUNG wire#w1
      Contact( "General Preparation"."Header 2"."CIP Request" )
   END_RUNG wire#w3
   // the same network as SCL:
   "CIP to Osa"."CIP Prep MB on Process" := "AlwaysTRUE" AND (("T-02_ChiliAwetan_1".Out_CIP_Req AND "CIP_to_Mix".CIP_RequestOK."Chili Awetan"."T-02.00_CIP_RequestOK") OR ("T-03_ChiliAwetan_2".Out_CIP_Req AND "CIP_to_Mix".CIP_RequestOK."Chili Awetan"."T-03.00_CIP_RequestOK") OR ("T-04_ChiliAwetan_3".Out_CIP_Req AND "CIP_to_Mix".CIP_RequestOK."Chili Awetan"."T-04.00_CIP_RequestOK") OR ("T-05_Tomato".Out_CIP_Req AND "CIP_to_Mix".CIP_RequestOK.Tomato."T-05.00_CIP_RequestOK") OR ("T-06_ChiliFresh_1".Out_CIP_Req AND "CIP_to_Mix".CIP_RequestOK.ChiliFresh."T-06.00_CIP_RequestOK") OR ("T-07_ChiliFresh_2".Out_CIP_Req AND "CIP_to_Mix".CIP_RequestOK.ChiliFresh."T-07.00_CIP_RequestOK") OR ("T-08_ChiliFresh_3".Out_CIP_Req AND "CIP_to_Mix".CIP_RequestOK.ChiliFresh."T-08.00_CIP_RequestOK") OR ("T-09_Garlic".Out_CIP_Req AND "CIP_to_Mix".CIP_RequestOK.Garlic."T-09.00_CIP_RequestOK") OR ("T-10_Vinegar".Out_CIP_Req AND "CIP_to_Mix".CIP_RequestOK.Vinegar."T-10.00_CIP_RequestOK") OR (("General Preparation"."Header 1"."CIP Request" OR "General Preparation"."Header 2"."CIP Request") AND "CIP_to_Mix".CIP_RequestOK.Header.Header_CIP_RequestOK));
END_REGION

REGION Network 39: OSA to CIP --- (CIP Request)
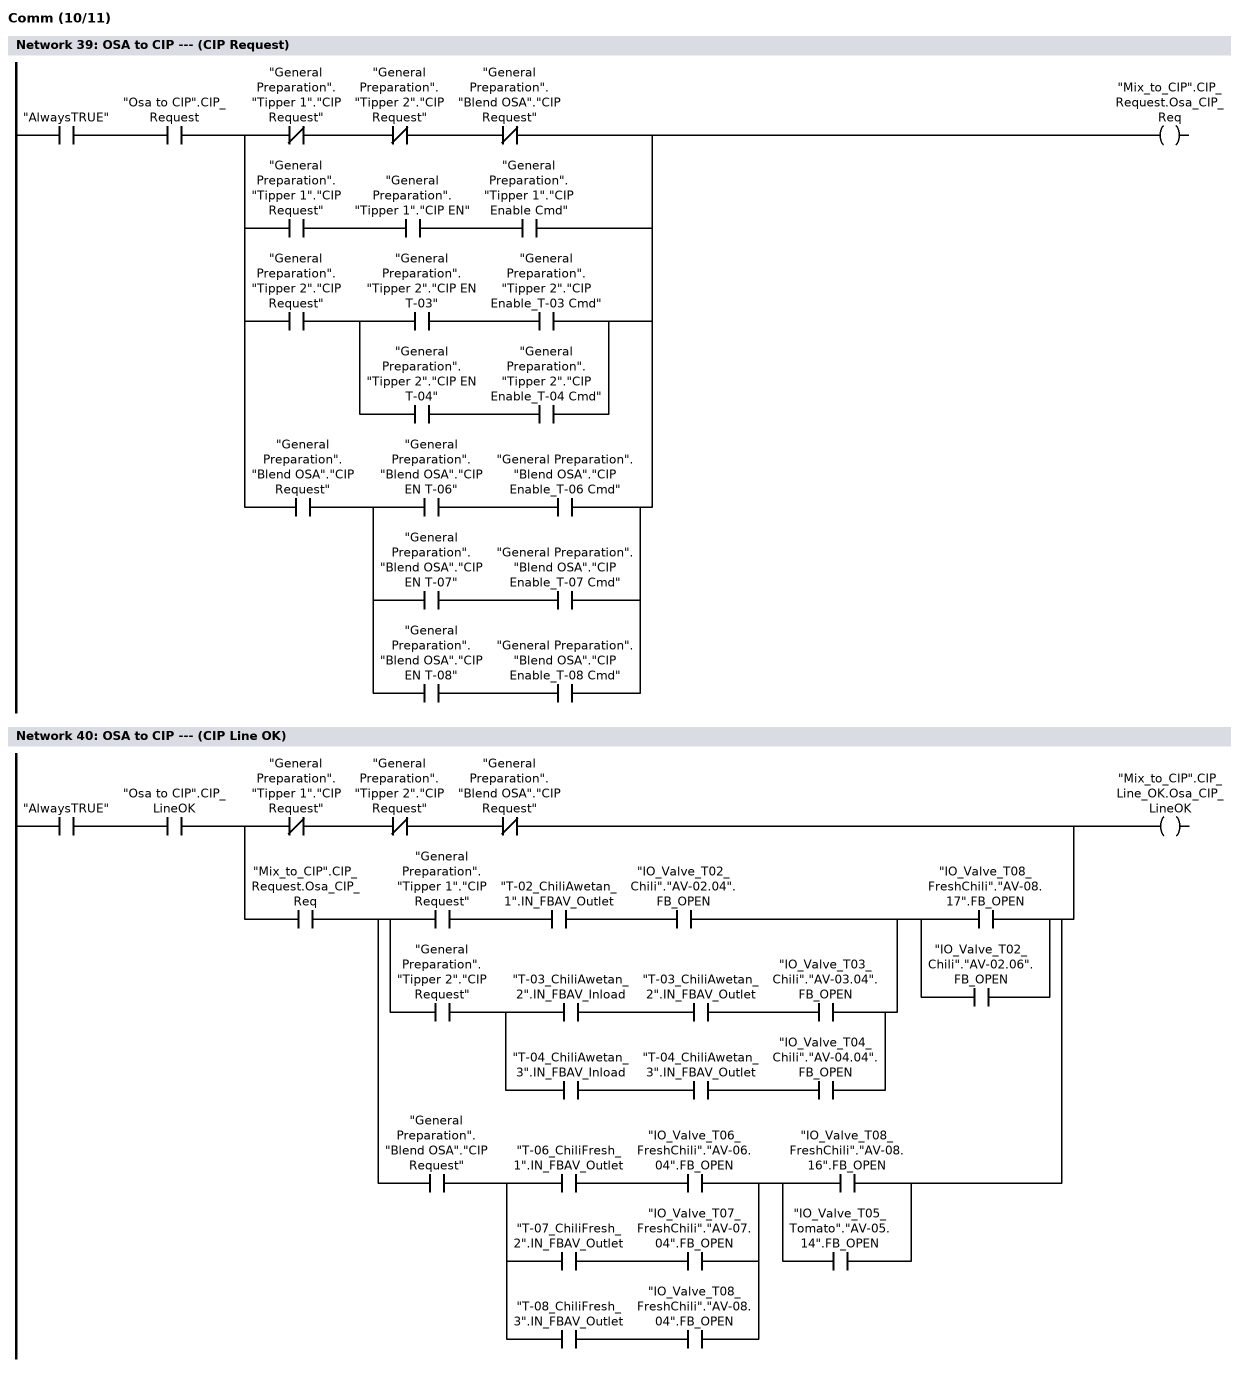
   RUNG wire#powerrail
      Contact( "AlwaysTRUE" )
      Contact( "Osa to CIP".CIP_Request )
      wire#w1
      I_Contact( "General Preparation"."Tipper 1"."CIP Request" )
      I_Contact( "General Preparation"."Tipper 2"."CIP Request" )
      I_Contact( "General Preparation"."Blend OSA"."CIP Request" )
      wire#w2
      Coil( "Mix_to_CIP".CIP_Request.Osa_CIP_Req )
   END_RUNG
   RUNG wire#w1
      Contact( "General Preparation"."Tipper 1"."CIP Request" )
      Contact( "General Preparation"."Tipper 1"."CIP EN" )
      Contact( "General Preparation"."Tipper 1"."CIP Enable Cmd" )
   END_RUNG wire#w2
   RUNG wire#w1
      Contact( "General Preparation"."Tipper 2"."CIP Request" )
      wire#w3
      Contact( "General Preparation"."Tipper 2"."CIP EN T-03" )
      Contact( "General Preparation"."Tipper 2"."CIP Enable_T-03 Cmd" )
   END_RUNG wire#w2
   RUNG wire#w3
      Contact( "General Preparation"."Tipper 2"."CIP EN T-04" )
      Contact( "General Preparation"."Tipper 2"."CIP Enable_T-04 Cmd" )
   END_RUNG wire#w2
   RUNG wire#w1
      Contact( "General Preparation"."Blend OSA"."CIP Request" )
      wire#w4
      Contact( "General Preparation"."Blend OSA"."CIP EN T-06" )
      Contact( "General Preparation"."Blend OSA"."CIP Enable_T-06 Cmd" )
   END_RUNG wire#w2
   RUNG wire#w4
      Contact( "General Preparation"."Blend OSA"."CIP EN T-07" )
      Contact( "General Preparation"."Blend OSA"."CIP Enable_T-07 Cmd" )
   END_RUNG wire#w2
   RUNG wire#w4
      Contact( "General Preparation"."Blend OSA"."CIP EN T-08" )
      Contact( "General Preparation"."Blend OSA"."CIP Enable_T-08 Cmd" )
   END_RUNG wire#w2
   // the same network as SCL:
   "Mix_to_CIP".CIP_Request.Osa_CIP_Req := "AlwaysTRUE" AND "Osa to CIP".CIP_Request AND ((NOT "General Preparation"."Tipper 1"."CIP Request" AND NOT "General Preparation"."Tipper 2"."CIP Request" AND NOT "General Preparation"."Blend OSA"."CIP Request") OR ("General Preparation"."Tipper 1"."CIP Request" AND "General Preparation"."Tipper 1"."CIP EN" AND "General Preparation"."Tipper 1"."CIP Enable Cmd") OR ("General Preparation"."Tipper 2"."CIP Request" AND (("General Preparation"."Tipper 2"."CIP EN T-03" AND "General Preparation"."Tipper 2"."CIP Enable_T-03 Cmd") OR ("General Preparation"."Tipper 2"."CIP EN T-04" AND "General Preparation"."Tipper 2"."CIP Enable_T-04 Cmd"))) OR ("General Preparation"."Blend OSA"."CIP Request" AND (("General Preparation"."Blend OSA"."CIP EN T-06" AND "General Preparation"."Blend OSA"."CIP Enable_T-06 Cmd") OR ("General Preparation"."Blend OSA"."CIP EN T-07" AND "General Preparation"."Blend OSA"."CIP Enable_T-07 Cmd") OR ("General Preparation"."Blend OSA"."CIP EN T-08" AND "General Preparation"."Blend OSA"."CIP Enable_T-08 Cmd"))));
END_REGION

REGION Network 40: OSA to CIP --- (CIP Line OK)
   RUNG wire#powerrail
      Contact( "AlwaysTRUE" )
      Contact( "Osa to CIP".CIP_LineOK )
      wire#w1
      I_Contact( "General Preparation"."Tipper 1"."CIP Request" )
      I_Contact( "General Preparation"."Tipper 2"."CIP Request" )
      I_Contact( "General Preparation"."Blend OSA"."CIP Request" )
      wire#w2
      Coil( "Mix_to_CIP".CIP_Line_OK.Osa_CIP_LineOK )
   END_RUNG
   RUNG wire#w1
      Contact( "Mix_to_CIP".CIP_Request.Osa_CIP_Req )
      wire#w3
      Contact( "General Preparation"."Tipper 1"."CIP Request" )
      Contact( "T-02_ChiliAwetan_1".IN_FBAV_Outlet )
      Contact( "IO_Valve_T02_Chili"."AV-02.04".FB_OPEN )
      wire#w4
      Contact( "IO_Valve_T08_FreshChili"."AV-08.17".FB_OPEN )
   END_RUNG wire#w2
   RUNG wire#w3
      Contact( "General Preparation"."Tipper 2"."CIP Request" )
      wire#w5
      Contact( "T-03_ChiliAwetan_2".IN_FBAV_Inload )
      Contact( "T-03_ChiliAwetan_2".IN_FBAV_Outlet )
      Contact( "IO_Valve_T03_Chili"."AV-03.04".FB_OPEN )
   END_RUNG wire#w4
   RUNG wire#w5
      Contact( "T-04_ChiliAwetan_3".IN_FBAV_Inload )
      Contact( "T-04_ChiliAwetan_3".IN_FBAV_Outlet )
      Contact( "IO_Valve_T04_Chili"."AV-04.04".FB_OPEN )
   END_RUNG wire#w4
   RUNG wire#w4
      Contact( "IO_Valve_T02_Chili"."AV-02.06".FB_OPEN )
   END_RUNG wire#w2
   RUNG wire#w3
      Contact( "General Preparation"."Blend OSA"."CIP Request" )
      wire#w6
      Contact( "T-06_ChiliFresh_1".IN_FBAV_Outlet )
      Contact( "IO_Valve_T06_FreshChili"."AV-06.04".FB_OPEN )
      wire#w7
      Contact( "IO_Valve_T08_FreshChili"."AV-08.16".FB_OPEN )
   END_RUNG wire#w2
   RUNG wire#w6
      Contact( "T-07_ChiliFresh_2".IN_FBAV_Outlet )
      Contact( "IO_Valve_T07_FreshChili"."AV-07.04".FB_OPEN )
   END_RUNG wire#w7
   RUNG wire#w6
      Contact( "T-08_ChiliFresh_3".IN_FBAV_Outlet )
      Contact( "IO_Valve_T08_FreshChili"."AV-08.04".FB_OPEN )
   END_RUNG wire#w7
   RUNG wire#w7
      Contact( "IO_Valve_T05_Tomato"."AV-05.14".FB_OPEN )
   END_RUNG wire#w2
   // the same network as SCL:
   "Mix_to_CIP".CIP_Line_OK.Osa_CIP_LineOK := "AlwaysTRUE" AND "Osa to CIP".CIP_LineOK AND ((NOT "General Preparation"."Tipper 1"."CIP Request" AND NOT "General Preparation"."Tipper 2"."CIP Request" AND NOT "General Preparation"."Blend OSA"."CIP Request") OR ("Mix_to_CIP".CIP_Request.Osa_CIP_Req AND (((("General Preparation"."Tipper 1"."CIP Request" AND "T-02_ChiliAwetan_1".IN_FBAV_Outlet AND "IO_Valve_T02_Chili"."AV-02.04".FB_OPEN) OR ("General Preparation"."Tipper 2"."CIP Request" AND (("T-03_ChiliAwetan_2".IN_FBAV_Inload AND "T-03_ChiliAwetan_2".IN_FBAV_Outlet AND "IO_Valve_T03_Chili"."AV-03.04".FB_OPEN) OR ("T-04_ChiliAwetan_3".IN_FBAV_Inload AND "T-04_ChiliAwetan_3".IN_FBAV_Outlet AND "IO_Valve_T04_Chili"."AV-04.04".FB_OPEN)))) AND ("IO_Valve_T08_FreshChili"."AV-08.17".FB_OPEN OR "IO_Valve_T02_Chili"."AV-02.06".FB_OPEN)) OR ("General Preparation"."Blend OSA"."CIP Request" AND (("T-06_ChiliFresh_1".IN_FBAV_Outlet AND "IO_Valve_T06_FreshChili"."AV-06.04".FB_OPEN) OR ("T-07_ChiliFresh_2".IN_FBAV_Outlet AND "IO_Valve_T07_FreshChili"."AV-07.04".FB_OPEN) OR ("T-08_ChiliFresh_3".IN_FBAV_Outlet AND "IO_Valve_T08_FreshChili"."AV-08.04".FB_OPEN)) AND ("IO_Valve_T08_FreshChili"."AV-08.16".FB_OPEN OR "IO_Valve_T05_Tomato"."AV-05.14".FB_OPEN)))));
END_REGION

REGION Network 41: CIP to OSA
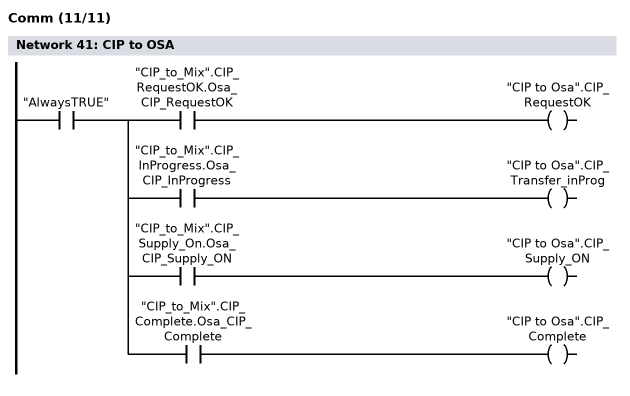
   RUNG wire#powerrail
      Contact( "AlwaysTRUE" )
      wire#w1
      Contact( "CIP_to_Mix".CIP_RequestOK.Osa_CIP_RequestOK )
      Coil( "CIP to Osa".CIP_RequestOK )
   END_RUNG
   RUNG wire#w1
      Contact( "CIP_to_Mix".CIP_InProgress.Osa_CIP_InProgress )
      Coil( "CIP to Osa".CIP_Transfer_inProg )
   END_RUNG
   RUNG wire#w1
      Contact( "CIP_to_Mix".CIP_Supply_On.Osa_CIP_Supply_ON )
      Coil( "CIP to Osa".CIP_Supply_ON )
   END_RUNG
   RUNG wire#w1
      Contact( "CIP_to_Mix".CIP_Complete.Osa_CIP_Complete )
      Coil( "CIP to Osa".CIP_Complete )
   END_RUNG
   // the same network as SCL:
   "CIP to Osa".CIP_RequestOK := "AlwaysTRUE" AND "CIP_to_Mix".CIP_RequestOK.Osa_CIP_RequestOK;
   "CIP to Osa".CIP_Transfer_inProg := "AlwaysTRUE" AND "CIP_to_Mix".CIP_InProgress.Osa_CIP_InProgress;
   "CIP to Osa".CIP_Supply_ON := "AlwaysTRUE" AND "CIP_to_Mix".CIP_Supply_On.Osa_CIP_Supply_ON;
   "CIP to Osa".CIP_Complete := "AlwaysTRUE" AND "CIP_to_Mix".CIP_Complete.Osa_CIP_Complete;
END_REGION
END_FUNCTION
